PROGRAM MAIN

VAR

END_VAR

GEMMA();
WATER_TANKS();
AIS();
SAFETY();
Q1_MOTOR();
Q2_MOTOR();

END_PROGRAM

(* stored: Version 1.1.0.1, ProductVersion 3.1.0.26
   POU MAIN: Id {4243ffa1-1c68-4f3e-be95-ae41ec879a6f} *)
